FUNCTION_BLOCK FB_ActorStopVerticalCommand IMPLEMENTS I_Command
VAR
	refFlyingHoist : REFERENCE TO FB_FlyingHoist;
END_VAR

METHOD Execute
IF (__ISVALIDREF(THIS^.refFlyingHoist)) THEN
	THIS^.refFlyingHoist.StopVerticalCommand();
END_IF
END_METHOD

METHOD FB_init : BOOL
VAR_INPUT
	bInitRetains 	: BOOL; // if TRUE, the retain variables are initialized (warm start / cold start)
	bInCopyCode 	: BOOL;  // if TRUE, the instance afterwards gets moved into the copy code (online change)
	refFlyingHoist 	: REFERENCE TO FB_FlyingHoist;
END_VAR
IF (__ISVALIDREF(refFlyingHoist)) THEN
	THIS^.refFlyingHoist REF= refFlyingHoist;
ELSE
	THIS^.refFlyingHoist REF= 0;
END_IF
END_METHOD

END_FUNCTION_BLOCK

(* stored: Version 1.1.0.1, ProductVersion 3.1.4022.18
   POU FB_ActorStopVerticalCommand: Id {25e706f3-ce24-4558-8364-8b63fd2cf54d}, SpecialFunc None
   Method Execute: Id {9e8c37f1-fd0f-4c4d-b262-cddfa75fb0f3}
   Method FB_init: Id {2ca43a7b-ddcc-4a1c-8c43-82e3087fb163} *)
